PROGRAM BWPoly3
VAR
	a: DINT;
	b: DINT;
	c: DINT;
	tempo_2: LREAL;
	tempo_3: LREAL;
	torque_per_thousand: DINT;
END_VAR

IF (TRAJ.tempo = 0) THEN
	TRAJ.v_max_rpm_low	:= (UDINT_TO_LREAL(TRAJ.speed_selector_rpm) / MOTOR.GEAR_RATIO);
	TRAJ.periodo_ms 	:= (ABS(TRAJ.position_selector_deg) * 15 * 1000) / (8 * TRAJ.v_max_rpm_low * 6) ; // millisecondi
	TRAJ.delta_t 		:= 1 / (TRAJ.periodo_ms); 
	TRAJ.status			:= TRUE;
	
	torque_per_thousand := LREAL_TO_INT(TRAJ.torque_selector_Nm*1000/MOTOR.RATED_TORQUE_NM);
	a := -64 * torque_per_thousand;
	b := 96 * torque_per_thousand;
	c := -32 * torque_per_thousand;

END_IF

IF (TRAJ.status = TRUE) THEN
	tempo_2 := TRAJ.tempo * TRAJ.tempo;
	tempo_3 := tempo_2 * TRAJ.tempo;
	TRAJ.target_torque_per_thousand := LREAL_TO_INT(a * tempo_3 + b * tempo_2 + c * TRAJ.tempo)/3;
ELSE
	TRAJ.error := PLC_ERROR.TRAJ_NO_SETUP;
END_IF

END_PROGRAM

(* stored: Version 1.1.0.1, ProductVersion 3.1.4024.11
   POU BWPoly3: Id {c02d5538-cdcd-4430-acbf-b91199ad5a2d}, SpecialFunc None *)
